PROGRAM MAIN
VAR
END_VAR

END_PROGRAM

(* stored: Version 1.1.0.1, ProductVersion 3.1.0.36
   POU MAIN: Id {466abbeb-cfc9-4942-9b05-128e1592f7cc}, SpecialFunc None *)
